INTERFACE ITF_State

METHOD Cycle : BOOL
VAR_INPUT
END_VAR
END_METHOD

END_INTERFACE

(* stored: Version 1.1.0.1, ProductVersion 3.1.4024.11
   Itf ITF_State: Id {73b3f942-a0c3-4df4-88b6-e9f74409a57e}
   Method Cycle: Id {f1e61e48-796a-45f4-8de0-014ff6e5344c} *)
